FUNCTION_BLOCK SimpleInit (* Simple FB with init event and one algorithm *)
  (* Standard: 61499-1 *)
  (* Version 0.0, 2018-10-15, Peter Gsellmann, TU Wien/ACIN *)
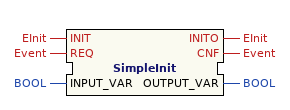
  EVENT_INPUT
    INIT : EInit; (* Init Request *)
    REQ; (* Normal Execution Request *)
  END_EVENT
  EVENT_OUTPUT
    INITO : EInit; (* Init Confirmation *)
    CNF; (* Execution Confirmation *)
  END_EVENT
  VAR_INPUT
    INPUT_VAR : BOOL; (* Input variable *)
  END_VAR
  VAR_OUTPUT
    OUTPUT_VAR : BOOL; (* Output variable *)
  END_VAR
  EC_STATES
    INIT : INIT -> INITO;
    REQ : REQ -> CNF;
  END_STATES
  ALGORITHM INIT IN ST:

  END_ALGORITHM
  ALGORITHM REQ IN ST:

  END_ALGORITHM
END_FUNCTION_BLOCK
